TYPE ST_CyCtrl ://气缸控制UDT  对应单控  双控气缸
STRUCT
   Io           : ST_CYIO;    //气缸IO
   Cmd      :  ST_CyCmd;
   Status     :ST_CyStatus;

END_STRUCT
END_TYPE

(* stored: Version 1.1.0.1, ProductVersion 3.1.4024.9
   DUT ST_CyCtrl: Id {551585b3-768c-49c4-a475-2377318c1d10} *)
